ABB RAPID module: Product2Mod.modx

MODULE Product2Mod



    PROC SeqProduct2()
        ProductPick;
        ProductProcess;
        ProductPlace;
    ENDPROC



    LOCAL PROC ProductPick()
        GripClose;
    ENDPROC



    LOCAL PROC ProductProcess()
        !
    ENDPROC



    LOCAL PROC ProductPlace()
        GripOpen;
    ENDPROC



    LOCAL PROC NotInUse()
    ENDPROC



ENDMODULE
